PROGRAM G7_Sel_Face
VAR_INPUT	
 SFCInit:BOOL;	
 SFCReset	:BOOL;

END_VAR

VAR
	Test_Face: BOOL;
END_VAR

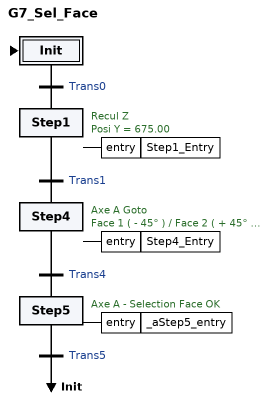
INITIAL_STEP Init:
END_STEP
TRANSITION FROM Init TO Step1
    := Trans0;
END_TRANSITION
// 										Recul Z
// Posi Y = 675.00
//
STEP Step1:
    Step1_Entry(P1);  // entry action
END_STEP
TRANSITION FROM Step1 TO Step4
    := Trans1;
END_TRANSITION
// 										Axe A Goto
// Face 1 ( - 45° ) / Face 2 ( + 45° )
// Ecretage ( + 90° )
//
STEP Step4:
    Step4_Entry(P1);  // entry action
END_STEP
TRANSITION FROM Step4 TO Step5
    := Trans4;
END_TRANSITION
// Axe A - Selection Face OK
STEP Step5:
    _aStep5_entry(P1);  // entry action
END_STEP
TRANSITION FROM Step5 TO Init
    := Trans5;
END_TRANSITION

ACTION _aStep5_entry:
Test_Face:=false;
END_ACTION

ACTION Step1_Entry:
Pos_cible_Y_Laser := 675;
En_pos_Y_Laser :=FALSE;
Top_Y_Laser := TRUE;

Pos_cible_Z_Laser := Pnc_axe_Z_Robot.Limite_Moins + 1;
En_pos_Z_Laser :=FALSE;
Top_Z_Laser := TRUE;
END_ACTION

ACTION Step4_Entry:
CASE Face_Cible OF
	1 : Pos_cible_A_Laser := 45;
	2 : Pos_cible_A_Laser := -45;
	3 : Pos_cible_A_Laser := -90;
END_CASE

En_pos_A_Laser :=FALSE;
Top_A_Laser := TRUE;

Face_En_Pos := FALSE;
END_ACTION

TRANSITION Trans0:
((Test_Face OR Auto) AND Top_Face )				
AND NOT Face_En_Pos 
AND Face_Cible <> 0 	
AND Face_Cible <> Face_En_Cours
END_TRANSITION

TRANSITION Trans1:
En_pos_Y_Laser AND NOT Top_Y_Laser AND En_pos_Z_Laser AND NOT Top_Z_Laser
END_TRANSITION

TRANSITION Trans4:
En_pos_A_Laser AND NOT Top_A_Laser 	AND
(Test_Face OR 
Auto) 									AND
NOT Top_Face 							AND
Face_En_Pos 							AND
Face_Cible <> 0 							AND
Face_Cible = Face_En_Cours
END_TRANSITION

TRANSITION Trans5:
NOT Top_Face 				AND
Face_En_Pos 				AND
Face_Cible <> 0 				AND
Face_Cible = Face_En_Cours
END_TRANSITION

END_PROGRAM

(* stored: Version 1.1.0.1
   POU G7_Sel_Face: Id {49dae811-3853-40e4-bac2-7b6e429e66a1}, SpecialFunc None
   Action _aStep5_entry: Id {f3cdd2f8-776c-4b9d-94f8-f1dda6a2c4ad}
   Action Step1_Entry: Id {ada27c39-3dc0-49b1-ad30-6a2eec0f2efa}
   Action Step4_Entry: Id {767f3cb6-ba5a-4a9c-9a41-c8a571a62f42}
   Transition Trans0: Id {04679d42-ab2b-466a-9504-c6066902e2e2}
   Transition Trans1: Id {5e2f641e-cdb8-479e-9a76-7524637eb271}
   Transition Trans4: Id {7e2007b4-2c2c-4787-88c8-f8f13a424ae0}
   Transition Trans5: Id {f9a130e9-d003-45a6-82ad-bbb2cf5a6791} *)
